{attribute 'linkalways'} 
{attribute 'no_explicit_call' := 'This FB is a CLASS and must be accessed using methods or properties'}
{attribute 'enable_dynamic_creation'}
FUNCTION_BLOCK FINAL GE_WORD EXTENDS Node
VAR
	in1 : _WORD(0);
	in2 : _WORD(0);
	out : _BOOL(FALSE);
END_VAR

METHOD PUBLIC Clone : I_Node
VAR
	pNode : POINTER TO GE_WORD;
END_VAR
pNode := __NEW(GE_WORD);
Clone := pNode^;
END_METHOD

METHOD FB_init : BOOL
VAR_INPUT
	bInitRetains : BOOL; // if TRUE, the retain variables are initialized (warm start / cold start)
	bInCopyCode : BOOL;  // if TRUE, the instance afterwards gets moved into the copy code (online change)
END_VAR
AddInput('in1',THIS^.in1);
AddInput('in2',THIS^.in2);
AddOutput('out', THIS^.out);
END_METHOD

METHOD PROTECTED OnExecute
VAR
END_VAR
out.Value := in1.Value >= in2.Value;
END_METHOD

END_FUNCTION_BLOCK

(* stored: Version 1.1.0.1, ProductVersion 3.1.4024.15
   POU GE_WORD: Id {a34a8b0a-9b0c-4c10-9590-165c4cfd355f}, SpecialFunc None
   Folder Constructor: Id {e92fa1bd-712e-47d0-9b72-a48f862a0f52}
   Method Clone: Id {941742e1-77a2-4f16-be4d-da24d7e76eac}
   Method FB_init: Id {30c8c7f1-b326-4eac-b34f-13c3388c101a}
   Method OnExecute: Id {e907f863-14a0-4a62-92c8-ad1fb963366d} *)
